Omron Sysmac Studio project PCEnvíaRecibe_2 (Sysmac Studio 1.23.0.14, StandardProject)

# Controller new_Controller_0: NX1P2-1040DT1 version 1.18
Task PrimaryTask (priority 4, period or condition 2000): Programa0

VAR_GLOBAL
    Mi_Puerto : _sDEVICE_PORT;
END_VAR
VAR_GLOBAL CONSTANT
    Mi_Modulo485 : _sOPTBOARD_ID := (SlotNo := 2, IPAdr := [5(16#0)]);
END_VAR
VAR_GLOBAL
    MiBufKind : _eSERIAL_BUF_KIND := _BUF_SENDRCV;
    Configuracion_Trama_Entrante : _sSERIAL_CFG;
    Orden_Leer : BOOL;
    Dato : ARRAY[0..1] OF BYTE;
    Dato_a_Enviar_Entrada0_ON : ARRAY[0..1] OF BYTE := [16#22, 16#33];
    Dato_a_Enviar_Entrada0_Off : ARRAY[0..1] OF BYTE := [16#7B, 16#5D];
    Dato_a_Enviar_Entrada1_ON : ARRAY[0..1] OF BYTE := [16#33, 16#44];
    Dato_a_Enviar_Entrada1_Off : ARRAY[0..1] OF BYTE := [16#8C, 16#6E];
    Dato_a_Enviar_Entrada2_ON : ARRAY[0..1] OF BYTE := [16#44, 16#55];
    Dato_a_Enviar_Entrada2_Off : ARRAY[0..1] OF BYTE := [16#9D, 16#7F];
    Valor_Sal_0_ON : ARRAY[0..1] OF BYTE := [16#34, 16#F2];
    Valor_Sal_0_OFF : ARRAY[0..1] OF BYTE := [16#25, 16#31];
    Valor_Sal_1_ON : ARRAY[0..1] OF BYTE := [16#22, 16#F1];
    Valor_Sal_1_OFF : ARRAY[0..1] OF BYTE := [16#11, 16#23];
    Sal_0 : BOOL;  (* at BuiltInIO://cpu/#0/Output_Bit_00 *)
    Sal_1 : BOOL;  (* at BuiltInIO://cpu/#0/Output_Bit_01 *)
    Numero_Bytes : UINT := 2;
    Ent_0 : BOOL;  (* Entrada 0; at BuiltInIO://cpu/#0/Input_Bit_00 *)
    Ent_1 : BOOL;  (* Entrada 1; at BuiltInIO://cpu/#0/Input_Bit_01 *)
    Ent_2 : BOOL;  (* Entrada 2; at BuiltInIO://cpu/#0/Input_Bit_02 *)
END_VAR

PROGRAM Programa0
VAR
    NX_SerialBufClear_Instance : NX_SerialBufClear;
    NX_SerialBufClear_Instance1 : NX_SerialBufClear;
    NX_SerialRcv_Instance1 : NX_SerialRcv;
    NX_SerialBufClear_Instance2 : NX_SerialBufClear;
    Instancia_NX_SerialSend1 : NX_SerialSend;
    Instancia_NX_SerialSend2 : NX_SerialSend;
    Instancia_NX_SerialSend3 : NX_SerialSend;
END_VAR
VAR_EXTERNAL
    Mi_Puerto : _sDEVICE_PORT;
END_VAR
VAR_EXTERNAL CONSTANT
    Mi_Modulo485 : _sOPTBOARD_ID;
END_VAR
VAR_EXTERNAL
    MiBufKind : _eSERIAL_BUF_KIND;
    Orden_Leer : BOOL;
    Dato : ARRAY[0..1] OF BYTE;
    Valor_Sal_0_ON : ARRAY[0..1] OF BYTE;
    Sal_0 : BOOL;
    Valor_Sal_0_OFF : ARRAY[0..1] OF BYTE;
    Sal_1 : BOOL;
    Valor_Sal_1_OFF : ARRAY[0..1] OF BYTE;
    Valor_Sal_1_ON : ARRAY[0..1] OF BYTE;
    Ent_0 : BOOL;
    Dato_a_Enviar_Entrada0_ON : ARRAY[0..1] OF BYTE;
    Numero_Bytes : UINT;
    Dato_a_Enviar_Entrada0_Off : ARRAY[0..1] OF BYTE;
    Ent_1 : BOOL;
    Dato_a_Enviar_Entrada1_ON : ARRAY[0..1] OF BYTE;
    Ent_2 : BOOL;
    Dato_a_Enviar_Entrada1_Off : ARRAY[0..1] OF BYTE;
    Dato_a_Enviar_Entrada2_ON : ARRAY[0..1] OF BYTE;
    Dato_a_Enviar_Entrada2_Off : ARRAY[0..1] OF BYTE;
    Configuracion_Trama_Entrante : _sSERIAL_CFG;
END_VAR
VAR
    _e1 : F_TRIG;
    _e2 : R_TRIG;
    _e3 : F_TRIG;
    _e4 : R_TRIG;
    _e5 : R_TRIG;
    _e6 : F_TRIG;
    _e7 : R_TRIG;
    _e8 : F_TRIG;
END_VAR

(* Section Recepción: ladder, written here as Structured Text *)

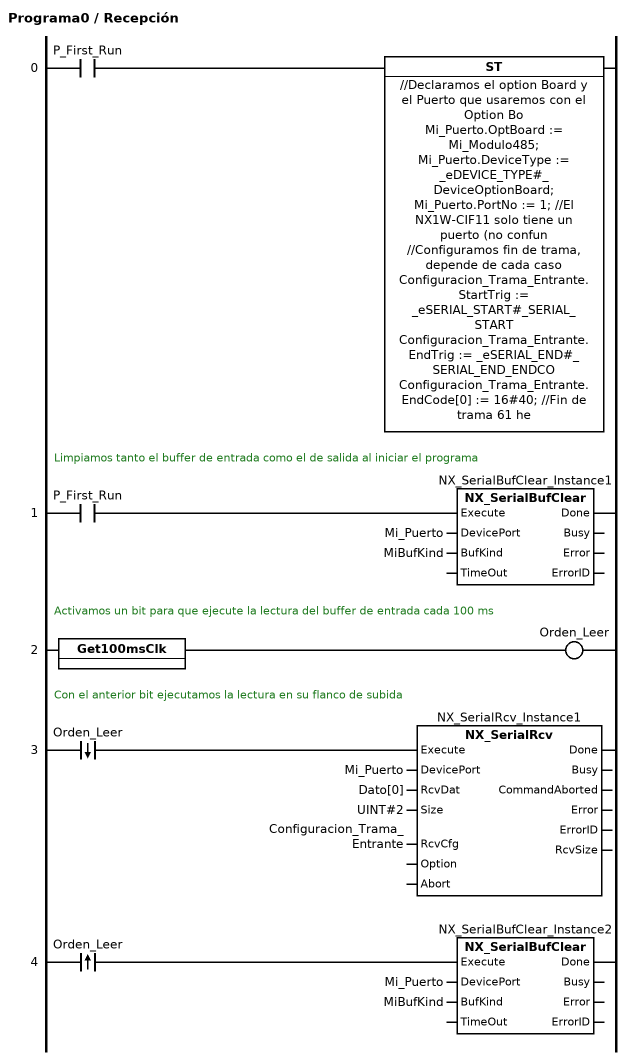
(* Rung 0 *)
IF P_First_Run THEN
    //Declaramos el option Board y el Puerto que usaremos con el Option Board anterior.
    Mi_Puerto.OptBoard := Mi_Modulo485;
    Mi_Puerto.DeviceType := _eDEVICE_TYPE#_DeviceOptionBoard;
    Mi_Puerto.PortNo := 1; //El NX1W-CIF11 solo tiene un puerto (no confundir con el slot donde está el módulo)
    
    //Configuramos fin de trama, depende de cada caso
    Configuracion_Trama_Entrante.StartTrig := _eSERIAL_START#_SERIAL_START_NONE; //No hay código de inicio
    Configuracion_Trama_Entrante.EndTrig := _eSERIAL_END#_SERIAL_END_ENDCODE1; //El final es marcado por cualquier byte
    Configuracion_Trama_Entrante.EndCode[0] := 16#40; //Fin de trama 61 hex '@'
END_IF;
(* Rung 1: Limpiamos tanto el buffer de entrada como el de salida al iniciar el programa *)
NX_SerialBufClear_Instance1(Execute := P_First_Run, DevicePort := Mi_Puerto, BufKind := MiBufKind);
(* Rung 2: Activamos un bit para que ejecute la lectura del buffer de entrada cada 100 ms *)
Orden_Leer := Get100msClk();
(* Rung 3: Con el anterior bit ejecutamos la lectura en su flanco de subida *)
_e1(CLK := Orden_Leer);
NX_SerialRcv_Instance1(Execute := _e1.Q, DevicePort := Mi_Puerto, RcvDat := Dato[0], Size := UINT#2, RcvCfg := Configuracion_Trama_Entrante);
(* Rung 4 *)
_e2(CLK := Orden_Leer);
NX_SerialBufClear_Instance2(Execute := _e2.Q, DevicePort := Mi_Puerto, BufKind := MiBufKind);

(* Section Salida: ladder, written here as Structured Text *)

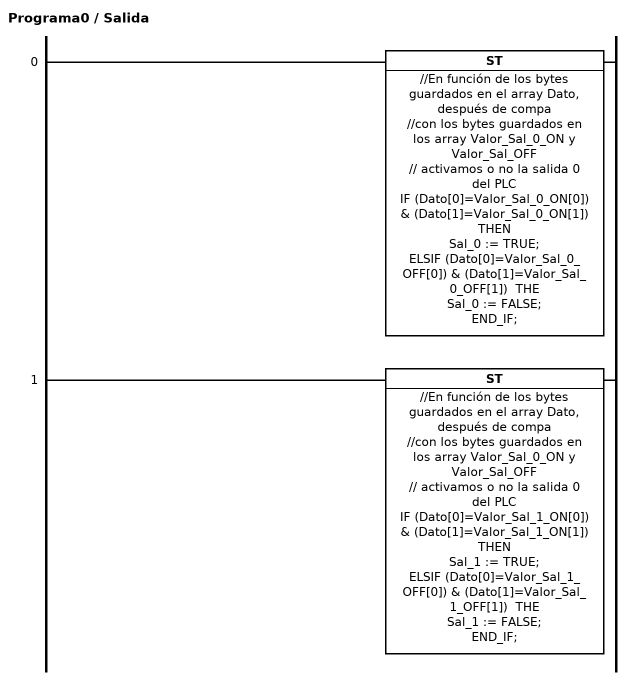
(* Rung 0 *)
//En función de los bytes guardados en el array Dato, después de compararlos
//con los bytes guardados en los array Valor_Sal_0_ON y Valor_Sal_OFF
// activamos o no la salida 0 del PLC
IF (Dato[0]=Valor_Sal_0_ON[0]) & (Dato[1]=Valor_Sal_0_ON[1]) THEN
    Sal_0 := TRUE;
ELSIF (Dato[0]=Valor_Sal_0_OFF[0]) & (Dato[1]=Valor_Sal_0_OFF[1])  THEN
	Sal_0 := FALSE;
END_IF;
(* Rung 1 *)
//En función de los bytes guardados en el array Dato, después de compararlos
//con los bytes guardados en los array Valor_Sal_0_ON y Valor_Sal_OFF
// activamos o no la salida 0 del PLC
IF (Dato[0]=Valor_Sal_1_ON[0]) & (Dato[1]=Valor_Sal_1_ON[1]) THEN
    Sal_1 := TRUE;
ELSIF (Dato[0]=Valor_Sal_1_OFF[0]) & (Dato[1]=Valor_Sal_1_OFF[1])  THEN
	Sal_1 := FALSE;
END_IF;

(* Section Envío: ladder, written here as Structured Text *)

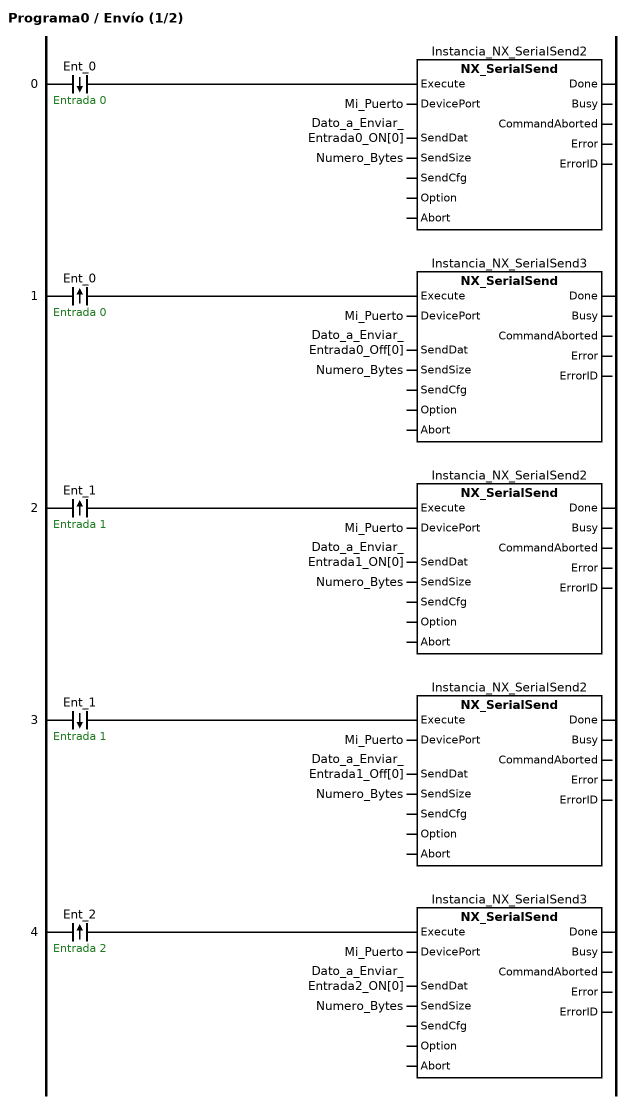
(* Rung 0 *)
_e3(CLK := Ent_0);
Instancia_NX_SerialSend2(Execute := _e3.Q, DevicePort := Mi_Puerto, SendDat := Dato_a_Enviar_Entrada0_ON[0], SendSize := Numero_Bytes);
(* Rung 1 *)
_e4(CLK := Ent_0);
Instancia_NX_SerialSend3(Execute := _e4.Q, DevicePort := Mi_Puerto, SendDat := Dato_a_Enviar_Entrada0_Off[0], SendSize := Numero_Bytes);
(* Rung 2 *)
_e5(CLK := Ent_1);
Instancia_NX_SerialSend2(Execute := _e5.Q, DevicePort := Mi_Puerto, SendDat := Dato_a_Enviar_Entrada1_ON[0], SendSize := Numero_Bytes);
(* Rung 3 *)
_e6(CLK := Ent_1);
Instancia_NX_SerialSend2(Execute := _e6.Q, DevicePort := Mi_Puerto, SendDat := Dato_a_Enviar_Entrada1_Off[0], SendSize := Numero_Bytes);
(* Rung 4 *)
_e7(CLK := Ent_2);
Instancia_NX_SerialSend3(Execute := _e7.Q, DevicePort := Mi_Puerto, SendDat := Dato_a_Enviar_Entrada2_ON[0], SendSize := Numero_Bytes);

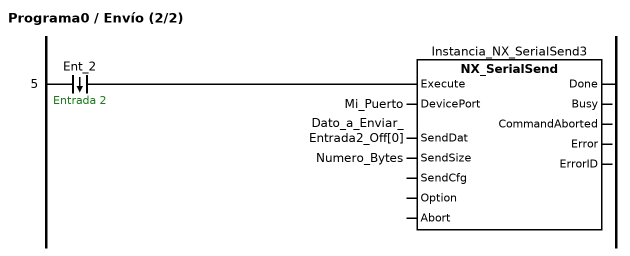
(* Rung 5 *)
_e8(CLK := Ent_2);
Instancia_NX_SerialSend3(Execute := _e8.Q, DevicePort := Mi_Puerto, SendDat := Dato_a_Enviar_Entrada2_Off[0], SendSize := Numero_Bytes);
END_PROGRAM